{attribute 'GeneratedUsingTerminal: IndraDrive MPB20-0003-0000'}
{attribute addProperty BoxType "IndraDrive MPB20-0003-0000"}
{attribute addProperty Id "AT_xAT %I*AT_x_475C3D7410MDTAT %Q*MDT_864618EC6WcStateAT %I*WcState_9091E0EB2InfoDataAT %I*InfoData_F60A43AC11"}
{attribute addProperty CRC "227280617"}
{attribute addProperty Size "29"}
TYPE IndraDrive_MPB20_0D8C06E9 EXTENDS TcoIo.EtcSlaveBoxBase_77A0E4A7 :
STRUCT
	{attribute addProperty Name "AT_x"}
	AT_x : AT_x_475C3D74;
	{attribute addProperty Name "MDT"}
	MDT : MDT_864618EC;
	{attribute addProperty Name "WcState"}
	WcState : TcoIo.WcState_9091E0EB;
	{attribute addProperty Name "InfoData"}
	InfoData : InfoData_F60A43AC;
END_STRUCT
END_TYPE

(* stored: Version 1.2.0.0, ProductVersion 3.1.4024.9
   DUT IndraDrive_MPB20_0D8C06E9: Id {a2f79ec8-3414-055a-3f07-28c32cf3a403} *)
